FUNCTION_BLOCK fb_temp_ctrl

VAR_INPUT
END_VAR

VAR_OUTPUT	
END_VAR

VAR
	separator_temp_dpi: fb_discrete_pi		:= (kc:=-4, ti:=15/60, Ts:=g_Ts_base, hi :=100, lo:=0, yout:=xmv_0[11]);	
	reactor_temp_dpi: fb_discrete_pi		:= (kc:=-8, ti:=7.5/60, Ts:=g_Ts_base, hi :=100, lo:=0, yout:=xmv_0[10]);
	
END_VAR

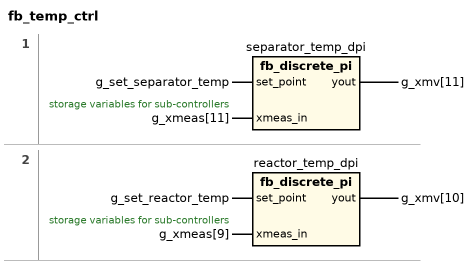
// NETWORK 1
//   g_xmeas[11]: storage variables for sub-controllers
separator_temp_dpi(set_point := g_set_separator_temp, xmeas_in := g_xmeas[11]); // fb_discrete_pi
g_xmv[11] := separator_temp_dpi.yout;

// NETWORK 2
//   g_xmeas[9]: storage variables for sub-controllers
reactor_temp_dpi(set_point := g_set_reactor_temp, xmeas_in := g_xmeas[9]); // fb_discrete_pi
g_xmv[10] := reactor_temp_dpi.yout;

END_FUNCTION_BLOCK

(* stored: Version 1.1.0.1, ProductVersion 3.1.0.26
   POU fb_temp_ctrl: Id {a76c6e58-1551-46ff-bf7f-b634b836a487} *)
